(* IEC 61131-3 sources: codefinetuner/third_party/tree-sitter-iec61131-3-st/examples, 13 files *)

(* ---- debouncer.st ---- *)
(*
 * Debouncer FB — filters a noisy boolean input by requiring it to stay
 * stable for `debounce_time` before reporting the new state.
 *)

FUNCTION_BLOCK Debounce
VAR_INPUT
    input         : BOOL;
    debounce_time : TIME := T#20ms;
END_VAR

VAR_OUTPUT
    output : BOOL;
END_VAR

VAR
    timer        : TON;
    pending      : BOOL;
END_VAR

(* Detect change, start the timer, latch the new value when stable. *)
IF input <> output THEN
    pending := TRUE;
    timer(IN := TRUE, PT := debounce_time);
    IF timer.Q THEN
        output := input;
        pending := FALSE;
        timer(IN := FALSE);
    END_IF
ELSE
    pending := FALSE;
    timer(IN := FALSE);
END_IF
END_FUNCTION_BLOCK

(* ---- edge-detector.st ---- *)
(*
 * Rising / falling edge detector — minimal R_TRIG / F_TRIG style FBs
 * implemented in ST.
 *)

FUNCTION_BLOCK RisingEdge
VAR_INPUT  CLK : BOOL; END_VAR
VAR_OUTPUT Q   : BOOL; END_VAR
VAR        prev : BOOL; END_VAR

Q := CLK AND NOT prev;
prev := CLK;
END_FUNCTION_BLOCK

FUNCTION_BLOCK FallingEdge
VAR_INPUT  CLK : BOOL; END_VAR
VAR_OUTPUT Q   : BOOL; END_VAR
VAR        prev : BOOL := FALSE; END_VAR

Q := NOT CLK AND prev;
prev := CLK;
END_FUNCTION_BLOCK

FUNCTION_BLOCK BothEdges
VAR_INPUT  CLK : BOOL; END_VAR
VAR_OUTPUT Q   : BOOL; END_VAR
VAR        prev : BOOL; END_VAR

Q := CLK <> prev;
prev := CLK;
END_FUNCTION_BLOCK

(* ---- lookup-table.st ---- *)
(*
 * Linear interpolation across a lookup table. Useful for sensor
 * linearization curves and gain schedulers.
 *)

TYPE
    LookupRow : STRUCT
        x : REAL;
        y : REAL;
    END_STRUCT;
END_TYPE

FUNCTION_BLOCK LookupTable
VAR_INPUT
    x          : REAL;
    table      : ARRAY [0..15] OF LookupRow;
    table_size : INT := 16;
    extrapolate : BOOL := FALSE;
END_VAR

VAR_OUTPUT
    y          : REAL;
    out_of_range : BOOL;
END_VAR

VAR
    i          : INT;
    span       : REAL;
    fraction   : REAL;
END_VAR

out_of_range := FALSE;

(* Below the first point. *)
IF x <= table[0].x THEN
    IF extrapolate AND table_size >= 2 THEN
        span := table[1].x - table[0].x;
        IF span > 0.0 THEN
            fraction := (x - table[0].x) / span;
            y := table[0].y + fraction * (table[1].y - table[0].y);
        ELSE
            y := table[0].y;
        END_IF
    ELSE
        y := table[0].y;
        out_of_range := x < table[0].x;
    END_IF
    RETURN;
END_IF

(* Above the last point. *)
IF x >= table[table_size - 1].x THEN
    IF extrapolate AND table_size >= 2 THEN
        span := table[table_size - 1].x - table[table_size - 2].x;
        IF span > 0.0 THEN
            fraction := (x - table[table_size - 2].x) / span;
            y := table[table_size - 2].y + fraction * (table[table_size - 1].y - table[table_size - 2].y);
        ELSE
            y := table[table_size - 1].y;
        END_IF
    ELSE
        y := table[table_size - 1].y;
        out_of_range := x > table[table_size - 1].x;
    END_IF
    RETURN;
END_IF

(* Find bracketing pair and linearly interpolate. *)
FOR i := 0 TO table_size - 2 DO
    IF x >= table[i].x AND x <= table[i + 1].x THEN
        span := table[i + 1].x - table[i].x;
        IF span > 0.0 THEN
            fraction := (x - table[i].x) / span;
            y := table[i].y + fraction * (table[i + 1].y - table[i].y);
        ELSE
            y := table[i].y;
        END_IF
        RETURN;
    END_IF
END_FOR
END_FUNCTION_BLOCK

(* ---- moving-average.st ---- *)
(*
 * N-sample circular-buffer moving average. Demonstrates ARRAY indexing,
 * MOD arithmetic, and instance-level state preservation.
 *)

FUNCTION_BLOCK MovingAverage
VAR_INPUT
    sample : REAL;
    reset  : BOOL;
END_VAR

VAR_OUTPUT
    average : REAL;
    full    : BOOL;
END_VAR

VAR CONSTANT
    WINDOW : INT := 16;
END_VAR

VAR
    buffer : ARRAY [0..15] OF REAL;
    head   : INT := 0;
    count  : INT := 0;
    sum    : REAL := 0.0;
    i      : INT;
END_VAR

IF reset THEN
    FOR i := 0 TO WINDOW - 1 DO
        buffer[i] := 0.0;
    END_FOR
    head := 0;
    count := 0;
    sum := 0.0;
    average := 0.0;
    full := FALSE;
    RETURN;
END_IF

(* Replace oldest sample, then advance the head pointer. *)
sum := sum - buffer[head] + sample;
buffer[head] := sample;
head := (head + 1) MOD WINDOW;

IF count < WINDOW THEN
    count := count + 1;
END_IF

average := sum / INT_TO_REAL(count);
full := count = WINDOW;
END_FUNCTION_BLOCK

(* ---- oop-shapes.st ---- *)
(*
 * OOP example — abstract Shape with concrete Circle and Rectangle, plus
 * a Drawable interface.
 *)

INTERFACE IDrawable
METHOD Draw : BOOL
END_METHOD
PROPERTY Color : DWORD
GET END_GET
SET END_SET
END_PROPERTY
END_INTERFACE

ABSTRACT FUNCTION_BLOCK Shape IMPLEMENTS IDrawable
VAR
    _color : DWORD := 16#FFFFFF;
END_VAR

METHOD ABSTRACT PUBLIC Area : REAL
END_METHOD

METHOD PUBLIC Draw : BOOL
    Draw := TRUE;
END_METHOD

PROPERTY PUBLIC Color : DWORD
GET
    Color := _color;
END_GET
SET
    _color := Color;
END_SET
END_PROPERTY
END_FUNCTION_BLOCK

FUNCTION_BLOCK Circle EXTENDS Shape
VAR_INPUT
    radius : REAL;
END_VAR

METHOD OVERRIDE PUBLIC Area : REAL
    Area := 3.14159 * radius * radius;
END_METHOD
END_FUNCTION_BLOCK

FUNCTION_BLOCK Rectangle EXTENDS Shape
VAR_INPUT
    width, height : REAL;
END_VAR

METHOD OVERRIDE PUBLIC Area : REAL
    Area := width * height;
END_METHOD
END_FUNCTION_BLOCK

(* ---- pid-controller.st ---- *)
(*
 * PID controller as a FUNCTION_BLOCK.
 *
 * Output = Kp*e + Ki*∫e dt + Kd*(de/dt), with anti-windup clamp on the
 * integral term.
 *)

FUNCTION_BLOCK PID
VAR_INPUT
    setpoint     : REAL;
    process_var  : REAL;
    Kp, Ki, Kd   : REAL;
    cycle_time   : TIME;
    out_min      : REAL := -100.0;
    out_max      : REAL :=  100.0;
    enable       : BOOL := TRUE;
END_VAR

VAR_OUTPUT
    output       : REAL;
END_VAR

VAR
    error        : REAL;
    prev_error   : REAL;
    integral     : REAL;
    derivative   : REAL;
    dt           : REAL;
END_VAR

IF NOT enable THEN
    integral := 0.0;
    output := 0.0;
    RETURN;
END_IF

dt := TIME_TO_REAL(cycle_time) / 1000.0;
error := setpoint - process_var;

(* Trapezoidal integration with anti-windup. *)
integral := integral + 0.5 * (error + prev_error) * dt;
IF integral > out_max THEN
    integral := out_max;
ELSIF integral < out_min THEN
    integral := out_min;
END_IF

IF dt > 0.0 THEN
    derivative := (error - prev_error) / dt;
ELSE
    derivative := 0.0;
END_IF

output := Kp * error + Ki * integral + Kd * derivative;
IF output > out_max THEN
    output := out_max;
ELSIF output < out_min THEN
    output := out_min;
END_IF

prev_error := error;
END_FUNCTION_BLOCK

(* ---- ramp-generator.st ---- *)
(*
 * Ramp generator — drives `output` from its current value toward
 * `target` with a fixed slope (units per second).
 *)

FUNCTION_BLOCK Ramp
VAR_INPUT
    target     : REAL;
    slope      : REAL := 10.0;       (* units per second *)
    cycle_time : TIME := T#10ms;
    enable     : BOOL := TRUE;
END_VAR

VAR_OUTPUT
    output : REAL;
    done   : BOOL;
END_VAR

VAR
    delta_per_cycle : REAL;
    diff            : REAL;
END_VAR

IF NOT enable THEN
    done := FALSE;
    RETURN;
END_IF

delta_per_cycle := slope * TIME_TO_REAL(cycle_time) / 1000.0;
diff := target - output;

IF ABS(diff) <= delta_per_cycle THEN
    output := target;
    done := TRUE;
ELSIF diff > 0.0 THEN
    output := output + delta_per_cycle;
    done := FALSE;
ELSE
    output := output - delta_per_cycle;
    done := FALSE;
END_IF
END_FUNCTION_BLOCK

(* ---- temperature-monitor.st ---- *)
(*
 * Temperature monitor — reads a sensor, scales raw counts to engineering
 * units, applies hysteresis, and triggers high/low alarms.
 *)

FUNCTION_BLOCK TempMonitor
VAR_INPUT
    raw_counts        : INT;
    raw_min, raw_max  : INT  := 0;
    eu_min,  eu_max   : REAL := 0.0;
    high_setpoint     : REAL;
    low_setpoint      : REAL;
    hysteresis        : REAL := 1.0;
END_VAR

VAR_OUTPUT
    temperature : REAL;
    high_alarm  : BOOL;
    low_alarm   : BOOL;
    in_range    : BOOL;
END_VAR

VAR
    span_raw : REAL;
    span_eu  : REAL;
END_VAR

(* Linear scaling. *)
span_raw := REAL_TO_LREAL(raw_max - raw_min);
span_eu  := eu_max - eu_min;
IF span_raw > 0.0 THEN
    temperature := eu_min + (REAL_TO_LREAL(raw_counts - raw_min) / span_raw) * span_eu;
ELSE
    temperature := eu_min;
END_IF

(* High alarm with hysteresis: trips at high_setpoint, clears at high_setpoint - hysteresis. *)
IF high_alarm THEN
    IF temperature < (high_setpoint - hysteresis) THEN
        high_alarm := FALSE;
    END_IF
ELSE
    IF temperature >= high_setpoint THEN
        high_alarm := TRUE;
    END_IF
END_IF

(* Low alarm with hysteresis. *)
IF low_alarm THEN
    IF temperature > (low_setpoint + hysteresis) THEN
        low_alarm := FALSE;
    END_IF
ELSE
    IF temperature <= low_setpoint THEN
        low_alarm := TRUE;
    END_IF
END_IF

in_range := NOT high_alarm AND NOT low_alarm;
END_FUNCTION_BLOCK

(* ---- blink.st ---- *)
(*
 * Blink — toggle an output at a fixed period using TON timers.
 *)

PROGRAM Blink
VAR
    on_timer  : TON;
    off_timer : TON;
    output    : BOOL;
    period_on  : TIME := T#500ms;
    period_off : TIME := T#500ms;
END_VAR

on_timer(IN := NOT output, PT := period_on);
off_timer(IN := output, PT := period_off);

IF on_timer.Q THEN
    output := TRUE;
END_IF

IF off_timer.Q THEN
    output := FALSE;
END_IF
END_PROGRAM

(* ---- configuration.st ---- *)
(*
 * Top-level CONFIGURATION / RESOURCE / TASK / PROGRAM mapping.
 * Demonstrates the IEC 61131-3 system architecture layer.
 *)

CONFIGURATION PlantConfig

VAR_GLOBAL
    g_emergency_stop : BOOL;
    g_total_uptime   : DINT;
END_VAR

RESOURCE Cpu1 ON CPU_001
    VAR_GLOBAL
        line1_state : INT;
    END_VAR

    TASK FastScan(INTERVAL := T#10ms, PRIORITY := 1);
    TASK SlowScan(INTERVAL := T#100ms, PRIORITY := 5);

    PROGRAM IO_Update     WITH FastScan : Conveyor;
    PROGRAM Coordinator   WITH SlowScan : PickAndPlace;
END_RESOURCE

RESOURCE Cpu2 ON CPU_002
    VAR_GLOBAL
        line2_state : INT;
    END_VAR

    TASK Periodic(INTERVAL := T#50ms, PRIORITY := 3);
    PROGRAM Hmi WITH Periodic : TempMonitor;
END_RESOURCE

END_CONFIGURATION

(* ---- conveyor.st ---- *)
(*
 * Conveyor with infeed/outfeed sensors, jam detection, and maintenance
 * counter.
 *)

PROGRAM Conveyor
VAR_INPUT
    start_button   : BOOL;
    stop_button    : BOOL;
    estop_button   : BOOL;
    infeed_sensor  : BOOL;
    outfeed_sensor : BOOL;
    motor_overload : BOOL;
END_VAR

VAR_OUTPUT
    motor_run      : BOOL;
    fault_lamp     : BOOL;
    parts_counted  : DINT;
END_VAR

VAR
    jam_timer       : TON;
    edge_outfeed    : R_TRIG;
    last_seen_part  : TIME;
    runtime_hours   : DINT;
    runtime_seconds : TON;
END_VAR

VAR CONSTANT
    JAM_TIMEOUT : TIME := T#10s;
END_VAR

(* E-stop and overload force shutdown immediately. *)
IF estop_button OR motor_overload THEN
    motor_run := FALSE;
    fault_lamp := TRUE;
    RETURN;
END_IF

(* Latch start/stop. *)
IF start_button AND NOT stop_button THEN
    motor_run := TRUE;
    fault_lamp := FALSE;
END_IF
IF stop_button THEN
    motor_run := FALSE;
END_IF

(* Jam detection: if the infeed sees a part but the outfeed never does. *)
jam_timer(IN := infeed_sensor AND NOT outfeed_sensor, PT := JAM_TIMEOUT);
IF jam_timer.Q THEN
    motor_run := FALSE;
    fault_lamp := TRUE;
END_IF

(* Count rising edges on the outfeed sensor. *)
edge_outfeed(CLK := outfeed_sensor);
IF edge_outfeed.Q THEN
    parts_counted := parts_counted + 1;
END_IF

(* Run-time counter — increments every hour the motor is on. *)
runtime_seconds(IN := motor_run, PT := T#1h);
IF runtime_seconds.Q THEN
    runtime_hours := runtime_hours + 1;
    runtime_seconds(IN := FALSE);
END_IF
END_PROGRAM

(* ---- state-machine.st ---- *)
(*
 * Sequential machine controller for a simple pick-and-place: HOME → DOWN →
 * GRIP → UP → MOVE → DOWN → RELEASE → UP → HOME.
 *)

TYPE
    Step : (
        HOME, MOVE_DOWN, GRIP, MOVE_UP, MOVE_OVER,
        DROP_DOWN, RELEASE, DROP_UP, RETURN_TO_HOME
    );
END_TYPE

PROGRAM PickAndPlace
VAR
    step : Step := HOME;
    cycle : DINT;
    z_axis_at_top, z_axis_at_bottom : BOOL;
    x_axis_at_pickup, x_axis_at_drop : BOOL;
    gripper_closed : BOOL;
    cmd_z_down, cmd_z_up : BOOL;
    cmd_x_to_drop, cmd_x_to_pickup : BOOL;
    cmd_grip_close, cmd_grip_open : BOOL;

    settle : TON;
END_VAR

CASE step OF
    HOME:
        IF z_axis_at_top AND x_axis_at_pickup THEN
            step := MOVE_DOWN;
        END_IF

    MOVE_DOWN:
        cmd_z_down := TRUE; cmd_z_up := FALSE;
        IF z_axis_at_bottom THEN
            cmd_z_down := FALSE;
            step := GRIP;
        END_IF

    GRIP:
        cmd_grip_close := TRUE;
        settle(IN := TRUE, PT := T#200ms);
        IF settle.Q THEN
            settle(IN := FALSE);
            gripper_closed := TRUE;
            step := MOVE_UP;
        END_IF

    MOVE_UP:
        cmd_z_up := TRUE;
        IF z_axis_at_top THEN
            cmd_z_up := FALSE;
            step := MOVE_OVER;
        END_IF

    MOVE_OVER:
        cmd_x_to_drop := TRUE;
        IF x_axis_at_drop THEN
            cmd_x_to_drop := FALSE;
            step := DROP_DOWN;
        END_IF

    DROP_DOWN:
        cmd_z_down := TRUE;
        IF z_axis_at_bottom THEN
            cmd_z_down := FALSE;
            step := RELEASE;
        END_IF

    RELEASE:
        cmd_grip_close := FALSE; cmd_grip_open := TRUE;
        settle(IN := TRUE, PT := T#200ms);
        IF settle.Q THEN
            settle(IN := FALSE);
            cmd_grip_open := FALSE;
            gripper_closed := FALSE;
            step := DROP_UP;
        END_IF

    DROP_UP:
        cmd_z_up := TRUE;
        IF z_axis_at_top THEN
            cmd_z_up := FALSE;
            step := RETURN_TO_HOME;
        END_IF

    RETURN_TO_HOME:
        cmd_x_to_pickup := TRUE;
        IF x_axis_at_pickup THEN
            cmd_x_to_pickup := FALSE;
            cycle := cycle + 1;
            step := HOME;
        END_IF
END_CASE
END_PROGRAM

(* ---- traffic-light.st ---- *)
(*
 * Traffic Light controller — single-intersection with NS / EW phases.
 *)

TYPE
    Phase : (NS_GREEN, NS_YELLOW, ALL_RED1, EW_GREEN, EW_YELLOW, ALL_RED2);
END_TYPE

PROGRAM TrafficLight
VAR
    state          : Phase := NS_GREEN;
    phase_timer    : TON;
    green_time     : TIME := T#15s;
    yellow_time    : TIME := T#3s;
    all_red_time   : TIME := T#1s;

    ns_red, ns_yellow, ns_green : BOOL;
    ew_red, ew_yellow, ew_green : BOOL;
END_VAR

CASE state OF
    NS_GREEN:
        ns_green := TRUE; ns_yellow := FALSE; ns_red := FALSE;
        ew_green := FALSE; ew_yellow := FALSE; ew_red := TRUE;
        phase_timer(IN := TRUE, PT := green_time);
        IF phase_timer.Q THEN
            phase_timer(IN := FALSE);
            state := NS_YELLOW;
        END_IF

    NS_YELLOW:
        ns_green := FALSE; ns_yellow := TRUE;
        phase_timer(IN := TRUE, PT := yellow_time);
        IF phase_timer.Q THEN
            phase_timer(IN := FALSE);
            state := ALL_RED1;
        END_IF

    ALL_RED1:
        ns_yellow := FALSE; ns_red := TRUE;
        phase_timer(IN := TRUE, PT := all_red_time);
        IF phase_timer.Q THEN
            phase_timer(IN := FALSE);
            state := EW_GREEN;
        END_IF

    EW_GREEN:
        ew_red := FALSE; ew_green := TRUE;
        phase_timer(IN := TRUE, PT := green_time);
        IF phase_timer.Q THEN
            phase_timer(IN := FALSE);
            state := EW_YELLOW;
        END_IF

    EW_YELLOW:
        ew_green := FALSE; ew_yellow := TRUE;
        phase_timer(IN := TRUE, PT := yellow_time);
        IF phase_timer.Q THEN
            phase_timer(IN := FALSE);
            state := ALL_RED2;
        END_IF

    ALL_RED2:
        ew_yellow := FALSE; ew_red := TRUE;
        phase_timer(IN := TRUE, PT := all_red_time);
        IF phase_timer.Q THEN
            phase_timer(IN := FALSE);
            state := NS_GREEN;
        END_IF
END_CASE
END_PROGRAM
